ABB RAPID module: Wizard.modx

MODULE Wizard
	PROC main()
		<SMT>
	ENDPROC
ENDMODULE
